FUNCTION_BLOCK FB_Hijo EXTENDS FB_Padre
VAR_INPUT
	iIn2:int;
END_VAR
VAR_OUTPUT
END_VAR
VAR
END_VAR

METHOD mMinus : INT
VAR_INPUT
	minus:INT;
END_VAR
mMinus := iIn1 - minus;
END_METHOD

METHOD mMultiply : INT
VAR_INPUT
END_VAR
//Hemos Sobreescrito el metodo del Padre. (superclase).

mMultiply:= THIS^.iIn1 * iIn2;
END_METHOD

METHOD mSuperMultiply : INT
VAR_INPUT
END_VAR
//Accedomos al metodo del padre con SUPER^.

mSuperMultiply := 10 * SUPER^.mMultiply();
END_METHOD

END_FUNCTION_BLOCK

(* stored: Version 1.1.0.1, ProductVersion 3.1.4024.12
   POU FB_Hijo: Id {6da2124f-b0d9-4aab-8349-c55f49aaee16}, SpecialFunc None
   Method mMinus: Id {392b875b-6247-4240-b383-b9d681cbef48}
   Method mMultiply: Id {c0cac5f4-ac9b-4744-8a26-90a08d49a4d4}
   Method mSuperMultiply: Id {17df23c8-9126-4208-95dd-6dbccaba4cc3} *)
